Fanuc KAREL source: CA0017.KL

PROGRAM CA0017
%STACKSIZE=65535
%PRIORITY=65535
%NOLOCKGROUP
TYPE
T=STRUCTURE
A : INTEGER
B : REAL
ENDSTRUCTURE
VAR
G : INTEGER
I : INTEGER
R : REAL
B : BOOLEAN
S : STRING[16]
AI : ARRAY[2] OF INTEGER
AR : ARRAY[2] OF REAL
ST : T
P : XYZWPR
V : VECTOR
ROUTINE F(P1 : INTEGER; P2 : INTEGER; P3 : INTEGER; P4 : INTEGER) FROM CA0017
ROUTINE F
BEGIN
G=(G + 1)
END F
BEGIN
G=0
I=1
R=2.5
B=TRUE
S='A'
AI[1]=3
AR[1]=4.5
-- UNSAFE_SOURCE_IR line 34: ST.A = 5
-- UNSAFE_SOURCE_IR line 35: ST.B = 6.5
F(I,I,I,I)
END CA0017
